KUKA KRL program: milling_1224_yuan22.src, milling_1224_yuan22.dat

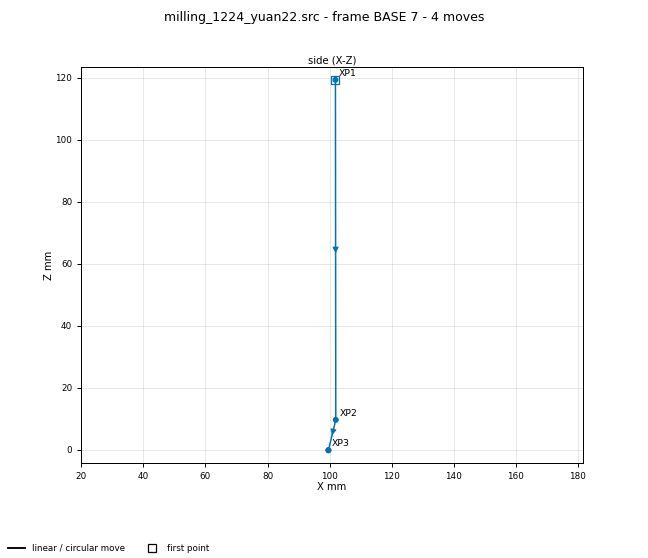
[picture p0: tool path of milling_1224_yuan22.src in frame BASE 7, 4 of 9 moves have a stored position in this frame; points joined in program order, loops and branches not executed]
--- milling_1224_yuan22.src ---
&ACCESS RVO
&REL 47
&PARAM EDITMASK = *
&PARAM TEMPLATE = C:\KRC\Roboter\Template\ExpertVorgabe
&PARAM DISKPATH = KRC:\R1\Program\zts1222
DEF milling_1224_yuan22( )


SpindleRun(TRUE,9000,#CLOCKWISE)

wait sec 1
pos_d=xp3

;FOLD PTP P1 CONT Vel=30 % PDAT1 Tool[6]:milling_8mm Base[7]:zts-1222;%{PE}
;FOLD Parameters ;%{h}
;Params IlfProvider=kukaroboter.basistech.inlineforms.movement.old; Kuka.IsGlobalPoint=False; Kuka.PointName=P1; Kuka.BlendingEnabled=True; Kuka.MoveDataPtpName=PDAT1; Kuka.VelocityPtp=30; Kuka.CurrentCDSetIndex=0; Kuka.MovementParameterFieldEnabled=True; IlfCommand=PTP
;ENDFOLD
$BWDSTART = FALSE
PDAT_ACT = PPDAT1
FDAT_ACT = FP1
BAS(#PTP_PARAMS, 30.0)
SET_CD_PARAMS (0)
PTP XP1 C_Dis
;ENDFOLD
;FOLD LIN P2 CONT Vel=0.1 m/s CPDAT1 Tool[6]:milling_8mm Base[7]:zts-1222 ;%{PE}
;FOLD Parameters ;%{h}
;Params IlfProvider=kukaroboter.basistech.inlineforms.movement.old; Kuka.IsGlobalPoint=False; Kuka.PointName=P2; Kuka.BlendingEnabled=True; Kuka.MoveDataName=CPDAT1; Kuka.VelocityPath=0.1; Kuka.CurrentCDSetIndex=0; Kuka.MovementParameterFieldEnabled=True; IlfCommand=LIN
;ENDFOLD
$BWDSTART = FALSE
LDAT_ACT = LCPDAT1
FDAT_ACT = FP2
BAS(#CP_PARAMS, 0.1)
SET_CD_PARAMS (0)
LIN XP2 C_Dis C_Dis
;ENDFOLD
;FOLD LIN P3 CONT Vel=0.01 m/s CPDAT2 Tool[6]:milling_8mm Base[7]:zts-1222 ;%{PE}
;FOLD Parameters ;%{h}
;Params IlfProvider=kukaroboter.basistech.inlineforms.movement.old; Kuka.IsGlobalPoint=False; Kuka.PointName=P3; Kuka.BlendingEnabled=True; Kuka.MoveDataName=CPDAT2; Kuka.VelocityPath=0.01; Kuka.CurrentCDSetIndex=0; Kuka.MovementParameterFieldEnabled=True; IlfCommand=LIN
;ENDFOLD
$BWDSTART = FALSE
LDAT_ACT = LCPDAT2
FDAT_ACT = FP3
BAS(#CP_PARAMS, 0.01)
SET_CD_PARAMS (0)
LIN XP3 C_Dis C_Dis
;ENDFOLD
$vel.cp=0.003
pos_d.z=pos_d.z-4
wait sec 0
$timer[1]=0
$timer_stop[1]=false
lin pos_d
x0_offset=pos_d.x
y0_offset=pos_d.y
z0_offset=pos_d.z
Rc=5.4
direc=true
if direc==true then
for ii=1 to 91
theta[ii]=(ii-1)*4.0
xy361[1,ii]=Rc*cos(theta[ii])+x0_offset
xy361[2,ii]=Rc*sin(theta[ii])+y0_offset
endfor
endif

;
x1_offset=pos_d.x
y1_offset=pos_d.y
z1_offset=pos_d.z
Rc1=2.7
direc=true
if direc==true then
for ii=1 to 91
theta1[ii]=(ii-1)*4.0
xy3611[1,ii]=Rc1*cos(theta1[ii])+x1_offset
xy3611[2,ii]=Rc1*sin(theta1[ii])+y1_offset
endfor
endif

;
cirp0.x=x0_offset
cirp0.y=y0_offset
cirp1.x=xy361[1,1]
cirp1.y=xy361[2,1]

cirp2.x=xy361[1,20]
cirp2.y=xy361[2,20]

cirp3.x=xy361[1,40]
cirp3.y=xy361[2,40]


cirp4.x=xy3611[1,65]
cirp4.y=xy3611[2,65]

cirp5.x=xy3611[1,20]
cirp5.y=xy3611[2,20]

$APO.CVEL=10
$vel.cp=0.003
;lin cirp1
lin pos_d
circ cirp4,cirp1,CA 180 c_vel
circ cirp2,cirp3,CA 361 c_vel
$vel.cp=0.01
lin pos_d
$timer_stop[1]=true

lin xp3
wait sec 1
SpindleRun(FALSE,0,#CLOCKWISE)
END

--- milling_1224_yuan22.dat ---
&ACCESS RVO
&REL 47
&PARAM EDITMASK = *
&PARAM TEMPLATE = C:\KRC\Roboter\Template\ExpertVorgabe
&PARAM DISKPATH = KRC:\R1\Program\zts1222
DEFDAT  milling_1224_yuan22 PUBLIC


DECL E6POS pos_u,pos_d,cirp,cirp0,cirp1,cirp2,cirp3,cirp4,cirp5,auxp1,auxp2
DECL BOOL direc
DECL REAL x0_offset,y0_offset,z0_offset,theta[91],xy361[2,361],xyz[3,6],Rc,A,B,Angle_x

DECL REAL x1_offset,y1_offset,z1_offset,theta1[91],xy3611[2,361],xyz1[3,6],Rc1,A1,B1,Angle_x1
DECL INT ii,jj,kk,Base_N
STRUC TUAN_TYP INT BASE_YUAN,REAL PHY



DECL E6POS XP1={X 101.901779,Y 31.1682568,Z 119.306831,A 47.4102631,B 0.121936962,C 0.0221000053,S 22,T 51,E1 0.0,E2 0.0,E3 0.0,E4 0.0,E5 0.0,E6 0.0}
DECL FDAT FP1={TOOL_NO 6,BASE_NO 7,IPO_FRAME #BASE,POINT2[] " "}
DECL PDAT PPDAT1={VEL 30.0000,ACC 100.000,APO_DIST 500.000,APO_MODE #CDIS,GEAR_JERK 100.000,EXAX_IGN 0}
DECL MODULEPARAM_T LAST_TP_PARAMS={PARAMS[] "Kuka.PointName=P3; Kuka.FrameData.base_no=7; Kuka.FrameData.tool_no=6; Kuka.FrameData.ipo_frame=#BASE; Kuka.isglobalpoint=False; Kuka.MoveDataPtpName=PDAT1; Kuka.MovementDataPdat.apo_mode=#CDIS; Kuka.MovementDataPdat.apo_dist=500; Kuka.MovementData.vel=0.01; Kuka.MovementData.acc=100; Kuka.MovementData.exax_ign=0; Kuka.VelocityPtp=30; Kuka.BlendingEnabled=True; Kuka.APXEnabled=False; Kuka.CurrentCDSetIndex=0; Kuka.FrameData.point2=; Kuka.MoveDataName=CPDAT2; Kuka.MovementData.apo_fac=50; Kuka.MovementData.apo_dist=500; Kuka.MovementData.axis_acc=100; Kuka.MovementData.axis_vel=100; Kuka.MovementData.circ_typ=#BASE; Kuka.MovementData.jerk_fac=50; Kuka.MovementData.ori_typ=#VAR; Kuka.VelocityPath=0.01                  "}
DECL E6POS XP2={X 102.014481,Y 31.0723705,Z 9.67388058,A 47.4097023,B 0.120903946,C 0.0214256328,S 22,T 51,E1 0.0,E2 0.0,E3 0.0,E4 0.0,E5 0.0,E6 0.0}
DECL FDAT FP2={TOOL_NO 6,BASE_NO 7,IPO_FRAME #BASE,POINT2[] " "}
DECL LDAT LCPDAT1={VEL 0.100000,ACC 100.000,APO_DIST 500.000,APO_FAC 50.0000,AXIS_VEL 100.000,AXIS_ACC 100.000,ORI_TYP #VAR,CIRC_TYP #BASE,JERK_FAC 50.0000,GEAR_JERK 100.000,EXAX_IGN 0}
DECL E6POS XP3={X 99.6330566,Y 31.0667896,Z -0.129563048,A 47.4096451,B 0.120777793,C 0.0215006713,S 22,T 51,E1 0.0,E2 0.0,E3 0.0,E4 0.0,E5 0.0,E6 0.0}
DECL FDAT FP3={TOOL_NO 6,BASE_NO 7,IPO_FRAME #BASE,POINT2[] " "}
DECL LDAT LCPDAT2={VEL 0.01000000,ACC 100.000,APO_DIST 500.000,APO_FAC 50.0000,AXIS_VEL 100.000,AXIS_ACC 100.000,ORI_TYP #VAR,CIRC_TYP #BASE,JERK_FAC 50.0000,GEAR_JERK 100.000,EXAX_IGN 0}
DECL E6POS XP4={X 1711.32727,Y 925.777039,Z 716.247620,A -42.1770058,B 0.00399478618,C 0.493762255,S 22,T 51,E1 0.0,E2 0.0,E3 0.0,E4 0.0,E5 0.0,E6 0.0}
DECL FDAT FP4={TOOL_NO 3,BASE_NO 25,IPO_FRAME #BASE,POINT2[] " "}
DECL LDAT LCPDAT3={VEL 0.300000,ACC 100.000,APO_DIST 500.000,APO_FAC 50.0000,AXIS_VEL 100.000,AXIS_ACC 100.000,ORI_TYP #VAR,CIRC_TYP #BASE,JERK_FAC 50.0000,GEAR_JERK 100.000,EXAX_IGN 0}
ENDDAT
